Staubli VAL3: page_trajectory.pjx

--- page_trajectory.pjx ---
Parameters version=s7.6.1 stackSize=5000 millimeterUnit=true
Program file=alreadyExist.pgx
Program file=buildList.pgx
Program file=cleanUserMenu.pgx
Program file=defineTraj.pgx
Program file=deleteItem.pgx
Program file=goTo.pgx
Program file=listAdd.pgx
Program file=loadPage.pgx
Program file=main.pgx
Program file=onEnterEvent.pgx
Program file=onExit.pgx
Program file=onF1Event.pgx
Program file=onF2Event.pgx
Program file=onF3Event.pgx
Program file=onF4Event.pgx
Program file=onF5Event.pgx
Program file=onF6Event.pgx
Program file=onF7Event.pgx
Program file=onF8Event.pgx
Program file=onLeftEvent.pgx
Program file=onRightEvent.pgx
Program file=onStart.pgx
Program file=refresh.pgx
Program file=refreshDynamic.pgx
Program file=refreshStatic.pgx
Program file=selectType.pgx
Program file=showStatus.pgx
Data file=page_trajectory.dtx
Library alias=trajType path=Disk://..//templates/trajectory/trajectory.pjx
Library alias=page path=Disk://kernel/template/page/page.pjx
Library alias=use path=Disk://kernel/userPage/userPage.pjx
Library alias=language path=Disk://kernel/language/language.pjx
Library alias=saveData path=Disk://saveData/saveData.pjx
Library alias=prog path=Disk://instruction/PROG/PROG.pjx
Library alias=cycleStatus path=Disk://cycleStatus/cycleStatus.pjx
Library alias=processList path=Disk://kernel/processList/processList.pjx
Library alias=OnEvent path=Disk://OnEvent/OnEvent.pjx
Library alias=tcp path=Disk://kernel/tool/tool.pjx
Type name=TrajectoryItem path=Disk://kernel/template/TrajectoryItem/TrajectoryItem.pjx
Type name=InstrItem path=Disk://kernel/template/InstrItem/InstrItem.pjx
Type name=FrameItem path=Disk://kernel/template/FrameItem/FrameItem.pjx

--- page_trajectory.dtx ---
num nIndex
num nKey = -1
public num nPage
num nRefresh = 2164.601
num nSelected
num nTime = 1
num nView
num nType
string sEvent = "hello"
string sEventImport
string sImport
public string sItems
string sList = "hello"
string sMenu[8]
  [0] = "Simulation"
  [4] = "Type"
  [5] = "Duplicate"
  [6] = "Delete"
  [7] = "New"
string sMenu8[8]
string sMenuUser[8]
string sMessage
bool bButton[8]
  [4] = true
  [5] = true
  [6] = true
  [7] = true
bool bLarge
num nIndexItem
num nOldIndex
bool bTrigger
num nClockStatus
bool bShowStatus
bool bMoveRelease

--- main.pgx ---
public program main()
  local bool l_bSave
  local bool l_bOverRide
  local bool l_bOk
  local bool l_bUnreached
  local string l_sMessage
begin
  // INIT
  call onStart()
  // LOOP UNTIL nKey=255
  nIndexItem=0
  do
    // GOTO
    call goTo(nIndexItem,l_bUnreached)
    if l_bUnreached
      // show the message out of range
      call language:message(l_sMessage,-5)
      call use:timerDialog(l_sMessage,1)
      l_bUnreached=false
    endIf
    call refresh()
    nKey=getKey()
    call use:listevent(nKey,nIndex,sEvent)
    nView=use:nView
    nSelected=nIndex
    //
    // OVERRIDE NORMAL FUNCTIONALITY-> POLYMORPHISM
    //
    if nKey>=271 and nKey<=278
      if sMenuUser[nKey-271]!=""
        // normal one
        call trajType:onFunctionSel(nIndex,sEvent,nKey)
        l_bOverRide=true
        call buildList()
        l_bSave=true
      endIf
    endIf
    if !l_bOverRide
      switch nKey
        case 264
          // left
          call onLeftEvent(l_bSave)
        break
        case 268
          // right
          call onRightEvent(l_bSave)
        break
        case 271
          // SIMULATION
          call onF1Event()
        break
        case 272
          // Option
          call onF2Event()
        break
        case 273
          call onF3Event()
        break
        case 274
          call onF4Event()
        break
        case 275
          // SELECT THE TRAJ TYPE
          call onF5Event()
        break
        case 276
          // DUPLICATE
          call onF6Event()
          l_bSave=true
        break
        case 277
          // DELETE
          call onF7Event()
          l_bSave=true
        break
        case 278
          // NEW
          call onF8Event()
          l_bSave=true
        break
        case 270
          call onEnterEvent()
        break
      endSwitch
    endIf
    l_bOverRide=false
    // release the resource
    delay(0)
    if nKey==255 and isKeyPressed(289)==true
      call language:message(l_sMessage,143)
      call use:timerDialog(l_sMessage,3)
    endIf
  until nKey==255 and isKeyPressed(289)==false
  // exit
  call onExit(l_bSave)
end

--- alreadyExist.pgx ---
program alreadyExist(string& x_sName[], bool& x_bUndo[])
  local num l_nX
  local num l_nY
  local string l_sString
begin
  // look if the trajectory already exist
  l_nX=40-use:nBottomX-1
  l_nY=use:nBottomY+1
  call language:message(l_sString,21)
  call use:type(l_nX,l_nY,l_sString)
  // read the new trajectory
  call use:read(l_nX+len(l_sString),l_nY,x_sName,10,false)
  if !use:bUseEscape
    call trajType:find(x_sName,x_bUndo)
    if x_bUndo
      call language:message(x_sName,-2)
      popUpMsg(x_sName)
    endIf
  else
    x_bUndo=true
  endIf
end

--- buildList.pgx ---
program buildList()
  local num l_nSize
  local string l_sEvent
  local num i
  local bool l_bFound
  local num l_nCount
  local string l_sEmpty
begin
  // INIT the list
  l_sEmpty=""
  call use:stringCopy(l_sEmpty,sList)
  // Build the list
  call trajType:getSize(l_nSize)
  for i=0 to l_nSize-1
    call trajType:get(l_sEvent,i)
    if l_sEvent!=""
      //
      // use the filter ?
      //
      // check if the bProcessList filter is active
      //
      l_bFound=true
      if saveData:sTrajFilter!=""
        l_bFound=find(l_sEvent,saveData:sTrajFilter)!=-1
      endIf
      // update the selected item
      if l_sEvent==sEvent
        nSelected=l_nCount
      endIf
      // add
      if l_bFound
        call listAdd(l_sEvent)
        l_nCount=l_nCount+1
      endIf
    endIf
  endFor
  // update
  use:bUseRefresh=true
end

--- cleanUserMenu.pgx ---
program cleanUserMenu()
  local num i
begin
  // clean all the reference
  for i=0 to size(sMenuUser)-1
    sMenuUser[i]=""
  endFor
end

--- defineTraj.pgx ---
program defineTraj()
  local num i
  local num l_nType
  local string l_sPath
begin
  // select the trajectory type
  if saveData:sTrajTypeUsing==""
    saveData:sTrajTypeUsing=saveData:sTrajType
  endIf
  // search inside all the instruction
  call saveData:getPathInstr(saveData:sTrajTypeUsing,l_sPath)
  // check the trajType
  if trajType:libPath()!=l_sPath and l_sPath!=""
    i=trajType:libLoad(l_sPath)
    delay(0)
  endIf
  // error
  if i!=0
    popUpMsg("error load traj type on ENTER"+saveData:sTrajTypeUsing+toString("",i))
  endIf
end

--- deleteItem.pgx ---
program deleteItem(bool& x_bResult)
  local string l_sSwap
  local num l_nResult
  local string l_sMessage
  local string l_sMessage2
  local bool l_bYes
  local string l_sButton[2]
  local InstrItem l_iSwap
begin
  //
  // delete a Trajectory
  //
  x_bResult=false
  // check
  if sEvent!=""
    l_iSwap.sType=saveData:sTrajTypeUsing
    l_iSwap.sData=sEvent
    call prog:findItem(l_iSwap,l_nResult,false)
    if l_nResult==0
      //delete it
      call language:message(l_sMessage,81)
      call language:getYesNo(l_sButton)
      // ask the yes_no question
      call use:yes_no(l_sMessage+"#"+saveData:sTrajTypeUsing+" "+sEvent,l_sButton,l_bYes)
      x_bResult=l_bYes
    endIf
  endIf
end

--- goTo.pgx ---
program goTo(num x_nIndex, bool& x_bUnreached[])
  local bool l_bUnreached
  local num l_nIndexTool
  local tool l_tTool
  local num l_nSize
  local string l_sItems[2]
  local num l_nId
  local num l_nResult
  local TrajectoryItem l_tTraj
begin
  // check the cycle status
  if !cycleStatus:bCycle and !cycleStatus:bSimulation
    // check the working Mode
    if cycleStatus:nWorkingMode==1 and isPowered()
      // set the memory for the moveHold button
      if cycleStatus:nWorkingStatus==6
        bMoveRelease=true
      endIf
      // check for the index
      if nOldIndex!=x_nIndex or (cycleStatus:nWorkingStatus!=0 and cycleStatus:nWorkingStatus!=6)
        if !isEmpty()
          resetMotion()
        endIf
        if nOldIndex!=x_nIndex
          nOldIndex=x_nIndex
        endIf
      else
        if isEmpty() and cycleStatus:nWorkingStatus==0 and bMoveRelease
          bMoveRelease=false
          cls()
          // copy the item to the trajectory
          l_sItems[0]=sEvent
          // take the elements
          call trajType:load(l_sItems,l_nResult)
          call trajType:getSizeItem(false,l_nSize)
          // MOVE
          do
            if x_nIndex>0
              call use:typeMenu(7,"<<")
            else
              call use:typeMenu(7,"    ")
            endIf
            if x_nIndex<=l_nSize
              call use:typeMenu(8,">>")
            else
              call use:typeMenu(8,"    ")
            endIf
            // get the data to move
            call trajType:getTool(l_nIndexTool)
            call tcp:getTool(l_tTool,l_nIndexTool)
            call trajType:getTrajItem(l_tTraj,x_nIndex)
            //
            // use a sTemp mdesc to set the blend off
            //
            l_tTraj.nom_speed.blend=off
            call trajType:goTo(l_tTool,l_tTraj.nom_speed,l_tTraj.moveType,x_bUnreached,x_nIndex)
            // TO DO language
            call use:timerDialog("Going to point: "+toString("",x_nIndex+1)+ " / "+toString("",l_nSize),0)
            do
              l_nId=getKey()
              call use:scroll(0,7,38,(getMoveId()-roundDown(getMoveId()))*100)
              delay(0)
            until isEmpty()or l_nId==255 or l_nId==277 or l_nId==278
            // continue
            if isEmpty() or (l_nId==278 and x_nIndex<l_nSize)
              if isEmpty()
                call use:timerDialog("At point: "+toString("",x_nIndex+1)+ " / "+toString("",l_nSize),1)
              endIf
              x_nIndex=x_nIndex+1
            elseIf l_nId==277 and x_nIndex>0
              // decrease
              x_nIndex=x_nIndex-1
            else
              delay(1)
            endIf
            // release
            resetMotion()
          until x_bUnreached or l_nId==255 or x_nIndex>=l_nSize or(x_nIndex==l_nSize and l_nSize==1)
          // refresh
          use:bUseRefresh=true
        endIf
      endIf
    else
      // reset the cycle
      if cycleStatus:nWorkingMode!=1 or !isPowered()
        resetMotion()
      endIf
    endIf
  endIf
  if l_nId==255
    // release
    call use:nullKey(l_nId)
  endIf
end

--- onEnterEvent.pgx ---
program onEnterEvent()
  local num i
  local num l_nIndex
  local string l_sItem[2]
  local num l_nResult
  local string l_sMessage
begin
  //
  // NB sEvent is the selected
  // element in the LIST
  //
  if sEvent!=""
    logMsg("Page trajectory trajtype "+trajType:libPath())
    //
    l_sItem=sEvent
    call trajType:onEdit(l_sItem)
    if find(l_sItem,"Disk://")!=-1 and l_nResult==0
      // load the page
      call loadPage(l_sItem,l_sItem[1])
    endIf
    // logMsg
    logMsg("[KERNEL] INTERFACE:PAGE Edit trajectory")
    //
    call buildList()
  endIf
  //
end

--- onExit.pgx ---
program onExit(bool x_bSave)
  local string l_sEmpty
  local num l_nResult
  local string l_sMessage
begin
  // resetMotion
  if !cycleStatus:bCycle
    resetMotion()
  endIf
  if x_bSave
    l_sEmpty=""
    l_nResult=0
    call trajType:onSave(l_sEmpty)
    // show the message
    call language:message(l_sMessage,-4)
    call use:timerDialog(l_sMessage,1)
  endIf
end

--- onF1Event.pgx ---
program onF1Event()
  local bool l_bYes
  local string l_sMessage
  local string l_sItem
  local num l_nResult
begin
  // look if the bButton is enable
  if bButton[0]
    //
    //SIMULATION
    //
    if !cycleStatus:bCycle and sEvent!=""
      // load the production page
      call loadPage("Disk://trajectory/page_simulation",sEvent)
      // save the moveHold
      bMoveRelease=false
    endIf
  endIf
end

--- onF2Event.pgx ---
program onF2Event()
  local string l_sMessage
  local string l_sEvent
  local string l_sFilter
  local num l_nIndex
  local num i
begin
  // look if the bButton is enable
  if bButton[1]
    //
    // make a selection list
    //
    // 0) Filter by name
    //
    call use:clear(0,13)
    call use:type(5,13,sMenu[1])
    call language:message(l_sMessage,85)
    call use:timerDialog(l_sMessage+": ",0)
    l_sFilter=saveData:sTrajFilter
    call use:read(20+(len(l_sMessage)/2)+1,5,l_sFilter,10,false)
    if !use:bUseEscape
      saveData:sTrajFilter=l_sFilter
    endIf

    // update
    call buildList()
    use:bUseRefresh=true
    // release the key
    call use:nullKey(nKey)
  endIf
end

--- onF3Event.pgx ---
program onF3Event()
begin
  // look if the bButton is enable
  if bButton[2]
    //
  endIf
end

--- onF4Event.pgx ---
program onF4Event()
  local string l_sMessage
  local bool l_bImport
  local string l_sPath[2]
  local num l_nLocal
  local num l_nKey
  local bool l_bDone
  local num l_nOldValue[4]
  local num i
  local num l_nDefault
  local string l_sButton[2]
  local string l_sItem
begin
  // look if the bButton is enable
  if bButton[3]
    //
  endIf
end

--- onF5Event.pgx ---
program onF5Event()
  local num i
  local num l_nValue
  local string l_sMessage
begin
  // look if the bButton is enable
  if bButton[4]
    //
    call selectType()
    //
    call buildList()
    //
    use:bUseRefresh=true
  endIf
end

--- onF6Event.pgx ---
program onF6Event()
  local string l_sPaste
  local bool l_bUndo
  local num l_nResult
begin
  // look if the bButton is enable
  if bButton[5]
    //
    //  Duplicate
    //
    l_sPaste=sEvent
    call alreadyExist(l_sPaste,l_bUndo)
    if !l_bUndo
      call trajType:duplicate(sEvent,l_sPaste,l_nResult)
      if l_nResult==0
        logMsg("[KERNEL] INTERFACE:Duplicate the trajectory: "+sEvent+" to: "+l_sPaste)
        sEvent=l_sPaste
        // update the memory stack
        call buildList()
      else
        popUpMsg("error code duplicate: "+toString("",l_nResult))
        logMsg("[KERNEL] INTERFACE:Duplicate the trajectory: "+sEvent+" to: "+l_sPaste+"errorCode"+toString("",l_nResult))
      endIf
    endIf
  endIf
end

--- onF7Event.pgx ---
program onF7Event()
  local string l_sSwap
  local num l_nResult
  local string l_sMessage
  local string l_sMessage2
  local bool l_bYes
  local string l_sButton[2]
begin
  // look if the bButton is enable
  if bButton[6]
    //
    // delete a Trajectory
    //
    call deleteItem(l_bYes)
    if l_bYes
      call trajType:delete(sEvent,l_nResult)
      if l_nResult==0
        logMsg("[KERNEL] INTERFACE:Delete the trajectory: "+saveData:sTrajTypeUsing+" "+sEvent)
        call buildList()
      else
        popUpMsg("error code: "+toString("",l_nResult))
        logMsg("[KERNEL] INTERFACE:Delete the trajectory: "+saveData:sTrajTypeUsing+" "+sEvent+"error code: "+toString("",l_nResult))
      endIf
    endIf
  endIf
end

--- onF8Event.pgx ---
program onF8Event()
  local string l_sNew
  local bool l_bUndo
  local num l_nResult
begin
  // look if the bButton is enable
  if bButton[7]
    // new one
    call alreadyExist(l_sNew,l_bUndo)
    if !l_bUndo and l_sNew!=""
      call trajType:new(l_sNew,l_nResult)
      if l_nResult==0
        logMsg("[KERNEL] INTERFACE:Create the new trajectory: "+saveData:sTrajTypeUsing+" "+l_sNew)
        sEvent=l_sNew
        call buildList()
      else
        popUpMsg("error code: "+toString("",l_nResult))
        logMsg("[KERNEL] INTERFACE:Create the new trajectory: "+saveData:sTrajTypeUsing+" "+l_sNew+" error code "+toString("",l_nResult))
      endIf
    endIf
  endIf
end

--- onLeftEvent.pgx ---
program onLeftEvent(bool& x_bSave)
  local num i
  local num l_nType
  local string l_sPath
  local string l_sEmpty
  local num l_nResult
  local string l_sMessage
begin
  // left click
  //
  //
  // select the previous one
  //
  if x_bSave
    x_bSave=false
    l_sEmpty=""
    l_nResult=0
    call trajType:onSave(l_sEmpty)
    // show the message
    call language:message(l_sMessage,-4)
    call use:timerDialog(l_sMessage,1)
  endIf
  // check it
  do
    nType=(nType+size(saveData:sTrajType)-1)%(size(saveData:sTrajType))
    saveData:sTrajTypeUsing=saveData:sTrajType[nType]
    if saveData:sTrajType[nType]!=""
      // find the good id
      call saveData:getPathInstr(saveData:sTrajType[nType],l_sPath)
    endIf
  until saveData:sTrajType[nType]!=""
  // load the type
  if trajType:libPath()!=l_sPath and l_sPath!=""
    i=trajType:libLoad(l_sPath)
    delay(0)
  endIf
  if l_sPath==""
    popUpMsg("error load traj type on ENTER "+saveData:sTrajTypeUsing+toString("",i))
  endIf
  // clean the user MENU
  call cleanUserMenu()
  // rebuild the list
  call buildList()
end

--- onRightEvent.pgx ---
program onRightEvent(bool& x_bSave)
  local num i
  local num l_nType
  local string l_sPath
  local string l_sEmpty
  local num l_nResult
  local string l_sMessage
begin
  //
  // right click
  //
  if x_bSave
    x_bSave=false
    l_sEmpty=""
    l_nResult=0
    call trajType:onSave(l_sEmpty)
    // show the message
    call language:message(l_sMessage,-4)
    call use:timerDialog(l_sMessage,1)
  endIf
  // select the next one
  do
    nType=(nType+1)%(size(saveData:sTrajType))
    saveData:sTrajTypeUsing=saveData:sTrajType[nType]
    if saveData:sTrajType[nType]!=""
      // find the good id
      if saveData:sTrajType[nType]!=""
        call saveData:getPathInstr(saveData:sTrajType[nType],l_sPath)
      endIf
    endIf
  until saveData:sTrajType[nType]!=""
  // load the type
  if trajType:libPath()!=l_sPath and l_sPath!=""
    i=trajType:libLoad(l_sPath)
    delay(0)
  endIf
  if l_sPath==""
    popUpMsg("error load traj type on ENTER "+saveData:sTrajTypeUsing+toString("",i))
  endIf
  // clean the user MENU
  call cleanUserMenu()
  // rebuild the list
  call buildList()
end

--- onStart.pgx ---
program onStart()
  local num i
begin
  // logMsg
  logMsg("[KERNEL] INTERFACE:PAGE Edit trajectory")
  // disable the filter
  if saveData:mode<2
    saveData:sTrajFilter=""
  endIf
  // check it
  if saveData:sTrajType[nType]!=saveData:sTrajTypeUsing
    for i=0 to size(saveData:sTrajType)-1
      // scan
      if saveData:sTrajTypeUsing==saveData:sTrajType[i]
        nType=i
        i=size(saveData:sTrajType)-1
      endIf
    endFor
  endIf
  // reset the Key pressure
  call use:nullKey(nKey)
  // define the select traj
  call defineTraj()
  // clean the userMenu
  call cleanUserMenu()
  // define the list
  call buildList()
end

--- refresh.pgx ---
program refresh()
// // page refresh
begin
  if !use:bShowDialog and !cycleStatus:bShowMessage
    // refresh the static message
    if (nKey>=270 and nKey<=278) or use:bUseRefresh
      call refreshStatic()
      call refreshDynamic()
    else
      // refresh the Dynamic message
      if abs(clock()-nRefresh)>nTime
        call refreshDynamic()
      endIf
    endIf
  endIf
  call showStatus()
  // release the resource
  delay(0)
end

--- refreshDynamic.pgx ---
program refreshDynamic()
  local string l_sMessage
begin
  // DO NOT CHANGE
  nRefresh=clock()
  use:bUseRefresh=false
  //
  // ADD HERE
  //
end

--- refreshStatic.pgx ---
program refreshStatic()
  local string l_sMessage
  local num i
begin
  cls()
  //
  // set the view of the page..
  //
  // SET THE PAGE NUMBER
  use:nPage=1010
  // USE <>PROFILE for <>PAGE
  use:nPage=use:nPage+abs(limit(saveData:mode,0,2)-2)
  if cycleStatus:bCycle
    use:nPage=use:nPage+3
  endIf
  // load the menu page
  if saveData:language!="japanese"
    // SET THE VIEW OF THE PAGE
    call language:page(l_sMessage,use:nPage)
    // define the menu
    call use:stringToArray(l_sMessage,sMenu)
  else
    // japanese use the array for the menu
    call language:page(sMenu8,use:nPage)
    call use:stringCopy(sMenu8,sMenu)
  endIf
  //
  // polymorphism
  //
  // get the user Menu or special one
  call trajType:getFunctionSel(sMenuUser)
  // OVERRIDE
  for i=0 to size(sMenuUser)-1
    if sMenuUser[i]!=""
      sMenu[i]=sMenuUser[i]
    endIf
  endFor
  // set the menu
  if saveData:language!="japanese"
    call use:setMenu(sMenu,true,3)
  else
    call use:setMenu(sMenu,false,3)
  endIf
  call use:getMenu(sMenu,bButton)
  //
  // CREATE THE LIST
  //
  // define your list size for default
  call use:setSizeList(19,0,19,11)
  call use:setView(bLarge)
  //
  call use:listcreate(saveData:sTrajTypeUsing)
  //
  call use:listadd(sList)
  //
  // refresh the list
  call use:selectNewField(nSelected,nIndex,nView)
  //
  // is a filter using ??
  if  saveData:sTrajFilter!=""
    call language:message(l_sMessage,64)
    call use:type(0,1,l_sMessage+">"+saveData:sTrajFilter)
  else
    // clean
    call use:typeLen(0,1," ",use:nBottomX)
  endIf
end

--- selectType.pgx ---
program selectType()
  local string l_sMessage
  local num l_nIndex
  local string l_sEvent
  local num l_nKey
  local num i
  local string l_sPath
begin
  // clean the line
  call use:clear(0,13)
  call language:message(l_sMessage,191)
  call use:typeCenter(13,l_sMessage,40,true)
  call use:setSizeList(15,2,10,6)
  // TODO message
  call use:listcreate("")
  call use:listadd(saveData:sTrajType)
  call use:selectNewField(nType,0,0)
  // select the Item
  do
    l_nKey=get()
    call use:listevent(l_nKey,l_nIndex,l_sEvent)
  until l_nKey==270 or l_nKey==255
  // choose the type
  if l_nKey==270 and saveData:sTrajTypeUsing!=l_sEvent
    saveData:sTrajTypeUsing=l_sEvent
    // get the path
    call saveData:getPathInstr(l_sEvent,l_sPath)
    // load it
    if trajType:libPath()!=l_sPath and l_sPath!=""
      i=trajType:libLoad(l_sPath)
      delay(0)
    endIf
    if l_sPath==""
      popUpMsg("error load traj type on ENTER "+saveData:sTrajTypeUsing+toString("",i))
    endIf
  endIf
  // clean the user MENU
  call cleanUserMenu()
end

--- showStatus.pgx ---
program showStatus()
  local joint l_jHere
  local point l_pHere
  local string l_sMessage[2]
  local tool l_tTool
  local num l_nIndexTool
  local frame l_fFrame
begin
  //
  // show an dialog box with
  // the current Joint/cartesian position
  //
  l_fFrame=world
  l_fFrame.trsf=saveData:fFrameItem[saveData:nFrameActive].fFrame.trsf
  call trajType:getTool(l_nIndexTool)
  call tcp:getTool(l_tTool,l_nIndexTool)
  if cycleStatus:nWorkingStatus>1 and cycleStatus:nWorkingStatus<5 and cycleStatus:nWorkingMode==1
    // set a timer of x second then the message disappear ..
    if !bTrigger
      nClockStatus=clock()
      bTrigger=true
      bShowStatus=true
    endIf
    if clock()-nClockStatus<saveData:nTimeDialog
      if cycleStatus:nWorkingStatus==2
        l_jHere=herej()
        l_sMessage="J1:"+toString("7.1",l_jHere.j1)
        l_sMessage=l_sMessage+"  J2:"+toString("7.1",l_jHere.j2)
        l_sMessage=l_sMessage+"  J3:"+toString("7.1",l_jHere.j3)+"#"
        l_sMessage=l_sMessage+"J4:"+toString("7.1",l_jHere.j4)
        l_sMessage=l_sMessage+"  J5:"+toString("7.1",l_jHere.j5)
        l_sMessage=l_sMessage+"  J6:"+toString("7.1",l_jHere.j6)
      else
        l_pHere=here(l_tTool,l_fFrame)
        l_sMessage="X :"+toString("7.1",l_pHere.trsf.x)
        l_sMessage=l_sMessage+"  Y :"+toString("7.1",l_pHere.trsf.y)
        l_sMessage=l_sMessage+"  Z :"+toString("7.1",l_pHere.trsf.z)+"#"
        l_sMessage=l_sMessage+"RX:"+toString("7.1",l_pHere.trsf.rx)
        l_sMessage=l_sMessage+"  RY:"+toString("7.1",l_pHere.trsf.ry)
        l_sMessage=l_sMessage+"  RZ:"+toString("7.1",l_pHere.trsf.rz)
      endIf
      call use:timerDialog(l_sMessage,0)
    else
      // disable it
      bShowStatus=false
    endIf
  else
    // reset it
    if bTrigger and !cycleStatus:bCycle
      resetMotion()
    endIf
    bTrigger=false
    bShowStatus=false
  endIf
end
